FUNCTION_BLOCK RecyclingFreezeProtection
VAR_INPUT
	CV: LREAL;
	Pressure: LREAL;
END_VAR
VAR_OUTPUT
	CV_OUT: LREAL;
END_VAR
VAR
	Hysteresis: Hysteresis;
END_VAR

Hysteresis(Value := Pressure, LimitValue := Main.GreenMaster.Parameters.Alarm.Limits.B.HeatExchangerHighPressure, Offset := 5);
IF Hysteresis.Above THEN
	CV_OUT := 0;
ELSE
	CV_OUT := CV;
END_IF

END_FUNCTION_BLOCK

(* stored: Version 1.1.0.1, ProductVersion 3.1.4024.6
   POU RecyclingFreezeProtection: Id {7fedce1a-72b8-4cfb-b806-53fb2d9609e3}, SpecialFunc None *)
